// TwinCAT 3 PLC project Pushover
// Title: Pushover
// Company: Stefan Besler
// Author: Stefan Besler and contributors
// ProjectVersion: 1.1.0
// ProgramVersion: 3.1.4023.0
// libraries:
//   Tc2_Standard, * (Beckhoff Automation GmbH)
//   Tc2_System, * (Beckhoff Automation GmbH)
//   Testbench, * (Zeugwerk GmbH)
// project tree:
//   / IPushoverClient.TcIO, PushoverClient.TcPOU
//   _DataTypes/ PushoverMessageType.TcDUT, PushoverPriority.TcDUT, PushoverRequest.TcDUT, PushoverSound.TcDUT
//   _Tests/ PushoverClientTest.TcPOU

// ---- _DataTypes/PushoverMessageType.TcDUT
{attribute 'qualified_only'}
{attribute 'strict'}
TYPE PushoverMessageType :
(
	Monospace := 0,
  Html
) INT;
END_TYPE

// ---- _DataTypes/PushoverPriority.TcDUT
{attribute 'qualified_only'}
{attribute 'strict'}
TYPE PushoverPriority :
(
  /// When the priority parameter is specified with a value of -2, messages will be considered lowest priority 
  /// and will not generate any notification. On iOS, the application badge number will be increased.
	Lowest := -2,
  
  /// Messages with a priority parameter of -1 will be considered low priority and will not generate any sound 
  /// or vibration, but will still generate a popup/scrolling notification depending on the client operating system. 
  /// Messages delivered during a user's quiet hours are sent as though they had a priority of (-1).
  Low := -1,
  
  /// Messages sent without a priority parameter, or sent with the parameter set to 0, will have the default priority. 
  /// These messages trigger sound, vibration, and display an alert according to the user's device settings. 
  /// On iOS, the message will display at the top of the screen or as a modal dialog, as well as in the notification center.
  /// On Android, the message will scroll at the top of the screen and appear in the notification center.
  ///
  /// If a user has quiet hours set and your message is received during those times, your message will be delivered as though it had a priority of -1.
  Normal := 0,
  
  /// Messages sent with a priority of 1 are high priority messages that bypass a user's quiet hours.
  /// These messages will always play a sound and vibrate (if the user's device is configured to) 
  /// regardless of the delivery time. High-priority should only be used when necessary and appropriate.
  /// 
  /// High-priority messages are highlighted in red in the device clients.
  High := 1,
  
  /// Emergency-priority notifications are similar to high-priority notifications, but they are repeated until the notification 
  /// is acknowledged by the user. These are designed for dispatching and on-call situations where it is critical that a 
  /// notification be repeatedly shown to the user (or all users of the group that the message was sent to) until it is acknowledged.
  /// The first user in a group to acknowledge a message will cancel retries for all other users in the group.
  ///
  /// Applications sending emergency notifications are issued a receipt that can be used to get the status of a notification and 
  /// find out whether it was acknowledged, or automatically receive a callback when the user has acknowledged the notification. 
  ///
  /// To send an emergency-priority notification, the priority parameter must be set to 2 and the retry and expire parameters must be supplied.
  ///
  /// The retry parameter specifies how often (in seconds) the Pushover servers will send the same notification to the user. 
  /// In a situation where your user might be in a noisy environment or sleeping, retrying the notification (with sound and vibration) 
  /// will help get his or her attention. This parameter must have a value of at least 30 seconds between retries.
  ///
  /// The expire parameter specifies how many seconds your notification will continue to be retried for (every retry seconds). 
  /// If the notification has not been acknowledged in expire seconds, it will be marked as expired and will stop being sent to the user. 
  /// Note that the notification is still shown to the user after it is expired, but it will not prompt the user for acknowledgement.
  /// This parameter must have a maximum value of at most 10800 seconds (3 hours), though the total number of retries will be capped at 50 regardless of the expire parameter.
  ///
  /// For example, sending a retry parameter of 60 and an expire parameter of 1800 will cause your notification to be retried
  /// every 60 seconds for 30 minutes. A retry parameter of 30 and an expire parameter of 10800 will retry every 30 seconds up to 25 minutes due to the cap of 50 retries.
  ///
  /// The optional callback parameter may be supplied with a publicly-accessible URL that pushover servers will 
  /// send a request to when the user has acknowledged your notification.
  /// When your application sends an emergency-priority notification, pushover API will respond with a receipt value that can be used to get information about
  /// whether the notification has been acknowledged. See pushover receipts and callbacks section for more information.
  /// If your application is not capable of storing receipt identifiers, you can send a tags parameter of comma-separated, arbitrary tags 
  /// which will be stored with the receipt on pushover servers. You can then use the cancel_by_tag API call to cancel all receipts with a specific tag.
  Emergency := 2
) INT;
END_TYPE

// ---- _DataTypes/PushoverRequest.TcDUT
TYPE INTERNAL PushoverRequest :
STRUCT
  TokenLength : INT;
  UserLength : INT;
  TitleLength : INT;  
  MessageLength : INT;
  DeviceLength : INT;
  UrlLength : INT;
  UrlTitleLength : INT;
  CallbackLength : INT;  
  ProxyHostLength : INT;  
  
  Retry : INT;
  Expire : INT;  
  MessageType : PushoverMessageType;  
  Priority : PushoverPriority;
  Sound : PushoverSound;
  Timestamp : INT; //< UNIX Timestamp in seconds 
  TimeToLive : INT; //< in seconds
  ProxyPort : INT;

  Token : STRING(80);
  User : STRING(80);  
  Device : STRING(80);
  Url : STRING(511);  
  UrlTitle : STRING(99);
  Callback : STRING(255);
  ProxyHost : STRING(80);
  Title : STRING(249);  
  Message : STRING(1023);  
END_STRUCT
END_TYPE

// ---- _DataTypes/PushoverSound.TcDUT
{attribute 'qualified_only'}
{attribute 'strict'}
TYPE PushoverSound :
(
  Pushover,
  Bike,
  Bugle,
  Cashregister,
  Classical,
  Cosmic,
  Falling,
  Gamelan,
  Incoming,
  Intermission,
  Magic,
  Mechanical,
  Pianobar,
  Siren,
  Spacealarm,
  Tugboat,
  Alien,
  Climb,
  Persistent_,
  Echo,
  Updown,
  Vibrate,
  None
) INT;
END_TYPE

// ---- IPushoverClient.TcIO
INTERFACE IPushoverClient

/// \copydoc Pushover.PushoverClient#Clear
METHOD Clear : IPushoverClient
END_METHOD

/// \copydoc Pushover.PushoverClient#EnableHtml
METHOD EnableHtml : IPushoverClient
END_METHOD

/// \copydoc Pushover.PushoverClient#EnableMonospace
METHOD EnableMonospace : IPushoverClient
END_METHOD

/// \copydoc Pushover.PushoverClient#SendMessageAsync
METHOD SendMessageAsync
VAR_IN_OUT CONSTANT
  title : STRING(255);
  message : STRING(255);
END_VAR
END_METHOD

/// \copydoc Pushover.PushoverClient#WithCallback
METHOD WithCallback : IPushoverClient
VAR_IN_OUT CONSTANT
  callback : STRING(255);
END_VAR
END_METHOD

/// \copydoc Pushover.PushoverClient#WithDevice
METHOD WithDevice : IPushoverClient
VAR_IN_OUT CONSTANT
  device : STRING(80);
END_VAR
END_METHOD

/// \copydoc Pushover.PushoverClient#WithExpire
METHOD WithExpire : IPushoverClient
VAR_INPUT
  expire : INT;
END_VAR
END_METHOD

/// \copydoc Pushover.PushoverClient#WithPriority
METHOD WithPriority : IPushoverClient
VAR_INPUT
  priority : PushoverPriority;
END_VAR
END_METHOD

/// \copydoc Pushover.PushoverClient#WithProxy
METHOD WithProxy : IPushoverClient
VAR_IN_OUT CONSTANT
  host : STRING(80);
END_VAR
VAR_INPUT
  port : INT;
END_VAR
END_METHOD

/// \copydoc Pushover.PushoverClient#WithRetry
METHOD WithRetry : IPushoverClient
VAR_INPUT
  retry : INT;
END_VAR
END_METHOD

/// \copydoc Pushover.PushoverClient#WithSound
METHOD WithSound : IPushoverClient
VAR_INPUT
  sound : PushoverSound;
END_VAR
END_METHOD

/// \copydoc Pushover.PushoverClient#WithTimestamp
METHOD WithTimestamp : IPushoverClient
VAR_INPUT
  timestamp : INT; //< UNIX Timestamp in seconds
END_VAR
END_METHOD

/// \copydoc Pushover.PushoverClient#WithTimeToLive
METHOD WithTimeToLive : IPushoverClient
VAR_INPUT
  ttl : INT; //< Seconds until this message should be automatically removed from the device. Needs to be positive
END_VAR
END_METHOD

/// \copydoc Pushover.PushoverClient#WithUrl
METHOD WithUrl : IPushoverClient
VAR_IN_OUT CONSTANT
  url : STRING(255);
END_VAR
END_METHOD

/// \copydoc Pushover.PushoverClient#WithUrlTitle
METHOD WithUrlTitle : IPushoverClient
VAR_IN_OUT CONSTANT
  urlTitle : STRING(255);
END_VAR
END_METHOD

END_INTERFACE

// ---- PushoverClient.TcPOU
/// This the main class of the library. It represents a Pushover app and
/// is tied to a unique API token. When constructing the object it is mandatory to pass
/// an `app-token` as well as a `user-token`.
///
/// Here's a simple example, which sends a pushover notification to a specific device of the user.
/// Note that this class uses a fluent API to configure the properties of a notification.
/// The actual action of sending the notification is triggered by [SendMessageAsync](xref:Pushover.PushoverClient#SendMessageAsync).
/// The ´Async´ Suffix in this method indicates that this action has to be waited for by checking for ´NOT _pushoverClient.Busy´ before
/// sending another notification.
///
/// ```sti
/// PROGRAM MAIN
/// VAR
///   _send : BOOL; // boolean, which can be triggered to send a message
///   _pushoverClient : Pushover.PushoverClient('<your_pushover_apptoken>', '<your_pushover_user>'); 
/// END_VAR
/// ```
/// ```std
/// IF _send
/// THEN
///   _send := FALSE;
///   _pushoverClient
///     .SendMessageAsync('Hello World!');
/// END_IF
///
/// _pushoverClient.Cyclic();
/// ```
{attribute 'conditionalshow_all_locals'}
{attribute 'no_explicit_call' := 'This FB is a CLASS and must be accessed using methods and/or properties'}
{attribute 'hide_all_locals'}
FUNCTION_BLOCK PushoverClient IMPLEMENTS IPushoverClient
VAR
  _busy : BOOL;
  _error : BOOL;
  _errorMessage : STRING(255);
  
  _request : PushoverRequest;
  _server : Tc2_System.ADSRDWRTEX;
END_VAR
VAR CONSTANT
  _defaultHost : STRING := '127.0.0.1.1.1';
  _defaultPort : UINT := 25733;
END_VAR

/// This property can be used to check if the client is ready for sending a notification. If the client is not 
/// ready or an error occurs during sending (e.g. not internet connection, Pushover Twincat Service is not running, ...)
/// the property [Error](xref:Pushover.PushoverClient#Error) returns `true`.
{attribute 'monitoring' := 'call'}
PROPERTY Busy : BOOL
GET
Busy := _busy;
END_GET
SET // PROTECTED
_busy := Busy;

IF _busy
THEN
  _error := FALSE;
END_IF
END_SET
END_PROPERTY

/// Resets all `WithXXX` statements to their default values.
METHOD Clear : IPushoverClient
VAR
  token : STRING;
  user : STRING;
  host : STRING := '127.0.0.1.1.1';
  port : UINT := 25733;  
END_VAR
token := THIS^.Token;
user := THIS^.User;
host := THIS^.Host;
port := THIS^.Port;

Tc2_System.MEMSET(ADR(_request), 0, SIZEOF(_request));
_request.Priority := PushoverPriority.Normal;
_request.Sound := PushoverSound.Pushover;

THIS^.Token := token;
THIS^.User := user;
THIS^.Host := _defaultHost;
THIS^.Port := _defaultPort;

Clear := THIS^;
END_METHOD

/// This method has to be called cyclically and takes care of the communication with the `Pushover Twincat Service`, which is reached 
/// via [Host](xref:Pushover.PushoverClient#Host) and [Port](xref:Pushover.PushoverClient#Port).
/// You can use the properties [Busy](xref:Pushover.PushoverClient#Busy) and [Error](xref:Pushover.PushoverClient#Error) to check weather an
/// operation was successful (`NOT Busy AND NOT Error`) or failed (`Error`), respectively.
METHOD Cyclic
VAR_INST
  errorTrig : Tc2_Standard.R_TRIG;
END_VAR
IF NOT Busy
THEN
  RETURN;
END_IF

_server(IDXOFFS:=0, 
        WRITELEN:=SIZEOF(_request),
        SRCADDR:=ADR(_request),
        WRTRD:=TRUE, 
        TMOUT:=T#5S,
        ERR=>,
        BUSY=>,
        ERRID=>);
  
IF _server.ERR // fallback to proxy
THEN
  Error := TRUE;
  ErrorMessage := Tc2_Standard.CONCAT('Error Code: ', UDINT_TO_STRING(_server.ERRID));
ELSIF NOT _server.BUSY 
THEN
  Busy := FALSE;
END_IF
END_METHOD

/// Enables Monospace in the pushover message
/// Either [HTML](xref:Pushover.PushoverClient#EnableHtml) or [Monospace](xref:Pushover.PushoverClient#EnableMonspace) can be enabled
METHOD EnableHtml : IPushoverClient
_request.MessageType := PushoverMessageType.Html;

EnableHtml := THIS^;
END_METHOD

/// Enables HTML in the pushover message
/// Either [HTML](xref:Pushover.PushoverClient#EnableHtml) or [Monospace](xref:Pushover.PushoverClient#EnableMonspace) can be enabled
METHOD EnableMonospace : IPushoverClient
_request.MessageType := PushoverMessageType.Monospace;

EnableMonospace := THIS^;
END_METHOD

/// Returns `true` if any error occured when calling an `XXX_Async` method of this object. The details of the error
/// are available by checking the proeprty
{attribute 'monitoring' := 'call'}
PROPERTY Error : BOOL
GET
Error := _error;
END_GET
SET // PROTECTED
_error := Error;

IF _error
THEN
  _busy := FALSE;
END_IF
END_SET
END_PROPERTY

/// Only valid if `Error=TRUE`, returns the explanation why the call of an `XXX_Async` method failed.
{attribute 'monitoring' := 'call'}
PROPERTY ErrorMessage : STRING(255)
GET
IF _error
THEN
  ErrorMessage := _errorMessage;
END_IF
END_GET
SET // PROTECTED
_errorMessage := ErrorMessage;
END_SET
END_PROPERTY

METHOD FB_init : BOOL
VAR_INPUT
	bInitRetains : BOOL; // if TRUE, the retain variables are initialized (warm start / cold start)
	bInCopyCode : BOOL;  // if TRUE, the instance afterwards gets moved into the copy code (online change)
  
  /// The pushover API token
  token : STRING;
  
  /// The user/group key (not e-mail address) of your user (or you),
  /// viewable when logged into the [pushover dashboard](https://pushover.net/login)
  user : STRING;
END_VAR
THIS^.Token := token;
THIS^.User := user;
THIS^.Host := _defaultHost;
THIS^.Port := _defaultPort;

Clear();
END_METHOD

/// Returns the AMS Net Id of the `Pushover Twincat Service`. Defauls to localhost
PROPERTY Host : STRING
GET
Host := _server.NETID;
END_GET
SET
_server(WRTRD := FALSE,
       NETID := Host,
       BUSY=>,
       ERR=>,
       ERRID=>);
END_SET
END_PROPERTY

PROPERTY Port : UINT
GET
Port := _server.PORT;
END_GET
SET
_server(WRTRD := FALSE,
       PORT := Port,
       BUSY=>,
       ERR=>,
       ERRID=>);
END_SET
END_PROPERTY

METHOD SendMessageAsync
VAR_IN_OUT CONSTANT
  title : STRING(255);
  message : STRING(255);
END_VAR
IF NOT Busy
THEN
  _request.TitleLength := Tc2_Standard.LEN(title);
  _request.Title := title;
  _request.MessageLength := Tc2_Standard.LEN(message);
  _request.Message := message;
  
  _server(WRTRD := FALSE,
         IDXGRP:=0,
         BUSY=>,
         ERR=>,
         ERRID=>);    
  Busy := TRUE;
ELSE
  Error := TRUE;
  _errorMessage := 'Client can not executed parallel requests!';
END_IF
END_METHOD

PROPERTY Token : STRING
GET
Token := _request.Token;
END_GET
SET
_request.Token := Token;
_request.TokenLength := Tc2_Standard.LEN(_request.Token);
END_SET
END_PROPERTY

PROPERTY User : STRING
GET
User := _request.User;
END_GET
SET
_request.User := User;
_request.UserLength := Tc2_Standard.LEN(_request.User);
END_SET
END_PROPERTY

/// Callback parameter may be supplied with a publicly-accessible URL that the
/// pushover servers will send a request to when the user has acknowledged your
/// notification.
/// Only used if priority is set to emergency.
METHOD WithCallback : IPushoverClient
VAR_IN_OUT CONSTANT
  callback : STRING(255);
END_VAR
_request.CallbackLength := Tc2_Standard.LEN(callback);
_request.Callback := callback;

WithCallback := THIS^;
END_METHOD

/// Your user's device name to send the message directly to that device,
/// rather than all of the user's devices
METHOD WithDevice : IPushoverClient
VAR_IN_OUT CONSTANT
  device : STRING(80);
END_VAR
_request.DeviceLength := Tc2_Standard.LEN(device);
_request.Device := device;

WithDevice := THIS^;
END_METHOD

/// Specifies how many seconds your notification will continue to be retried for (every retry seconds).
/// Only required if priority is set to emergency.
METHOD WithExpire : IPushoverClient
VAR_INPUT
  expire : INT;
END_VAR
_request.Expire := expire;

WithExpire := THIS^;
END_METHOD

/// Priority of the message
METHOD WithPriority : IPushoverClient
VAR_INPUT
  priority : PushoverPriority;
END_VAR
_request.Priority := priority;

WithPriority := THIS^;
END_METHOD

/// Adds a ttl to the Pushover message
METHOD WithProxy : IPushoverClient
VAR_IN_OUT CONSTANT
  host : STRING(80);
END_VAR
VAR_INPUT
  port : INT;
END_VAR
_request.ProxyHostLength := Tc2_Standard.LEN(host);
_request.ProxyHost := host;
_request.ProxyPort := port;

WithProxy := THIS^;
END_METHOD

/// Specifies how often (in seconds) the Pushover servers will send the same notification to the user.
/// Only required if priority is set to emergency.
METHOD WithRetry : IPushoverClient
VAR_INPUT
  retry : INT;
END_VAR
_request.Retry := retry;

WithRetry := THIS^;
END_METHOD

/// Priority of the message
METHOD WithSound : IPushoverClient
VAR_INPUT
  sound : PushoverSound;
END_VAR
_request.Sound := sound;

WithSound := THIS^;
END_METHOD

/// A Unix timestamp of your message's date and time to display to the user,
/// rather than the time your message is received by the pushover API
METHOD WithTimestamp : IPushoverClient
VAR_INPUT
  timestamp : INT; //< UNIX Timestamp in seconds
END_VAR
_request.Timestamp := timestamp;

WithTimestamp := THIS^;
END_METHOD

/// Adds a ttl to the Pushover message
METHOD WithTimeToLive : IPushoverClient
VAR_INPUT
  ttl : INT; //< Seconds until this message should be automatically removed from the device. Needs to be positive
END_VAR
_request.TimeToLive := ttl;

WithTimeToLive := THIS^;
END_METHOD

/// A supplementary URL to show with your message
METHOD WithUrl : IPushoverClient
VAR_IN_OUT CONSTANT
  url : STRING(255);
END_VAR
_request.UrlLength := Tc2_Standard.LEN(url);
_request.Url := url;

WithUrl := THIS^;
END_METHOD

/// A title for your supplementary URL, otherwise just the URL is shown
METHOD WithUrlTitle : IPushoverClient
VAR_IN_OUT CONSTANT
  urlTitle : STRING(255);
END_VAR
_request.UrlTitleLength := Tc2_Standard.LEN(urlTitle);
_request.UrlTitle := urlTitle;

WithUrlTitle := THIS^;
END_METHOD

END_FUNCTION_BLOCK

// ---- _Tests/PushoverClientTest.TcPOU
FUNCTION_BLOCK PushoverClientTest EXTENDS PushoverClient IMPLEMENTS Testbench.IUnitTest
VAR
  _sampleRequest : PushoverRequest;
END_VAR
VAR CONSTANT
  _testAppToken : STRING := 'APP_TOKEN';
  _testUserToken : STRING := 'USER_TOKEN';
END_VAR

METHOD FB_init : BOOL
VAR_INPUT
	bInitRetains : BOOL; // if TRUE, the retain variables are initialized (warm start / cold start)
	bInCopyCode : BOOL;  // if TRUE, the instance afterwards gets moved into the copy code (online change)
  
  /// The pushover API token
  token : STRING;
  
  /// The user/group key (not e-mail address) of your user (or you),
  /// viewable when logged into the [pushover dashboard](https://pushover.net/login)
  user : STRING;
END_VAR
SUPER^.FB_init(bInitRetains, bInCopyCode, _testAppToken, _testUserToken);

_sampleRequest.TokenLength := 1;
_sampleRequest.UserLength := 2;
_sampleRequest.TitleLength := 3;
_sampleRequest.MessageLength := 4;
_sampleRequest.DeviceLength := 5;
_sampleRequest.UrlLength := 6;
_sampleRequest.UrlTitleLength := 7;
_sampleRequest.CallbackLength := 8;
_sampleRequest.ProxyHostLength := 9;
  
_sampleRequest.Token := 'token';
_sampleRequest.User := 'user';
_sampleRequest.Retry := 3;
_sampleRequest.Expire := 5;
_sampleRequest.MessageType := PushoverMessageType.Html;  
_sampleRequest.Priority := PushoverPriority.High;
_sampleRequest.Sound := PushoverSound.Cashregister;
_sampleRequest.Timestamp := 5;
_sampleRequest.TimeToLive := 50;
_sampleRequest.ProxyPort := 8080;

_sampleRequest.Title := 'Title';
_sampleRequest.Message := 'Message';
_sampleRequest.Device := 'Device';
_sampleRequest.Url := 'Url';
_sampleRequest.UrlTitle := 'UrlTitle';
_sampleRequest.Callback := 'Callback';
_sampleRequest.ProxyHost := 'ProxyHost';
END_METHOD

METHOD SendMessageAsync
VAR_IN_OUT CONSTANT
  title : STRING(255);
  message : STRING(255);
END_VAR
IF NOT Busy
THEN
  _request.TitleLength := Tc2_Standard.LEN(title);
  _request.Title := title;
  _request.MessageLength := Tc2_Standard.LEN(message);
  _request.Message := message;
  
  _server(WRTRD := FALSE,
         IDXGRP:=0,
         BUSY=>,
         ERR=>,
         ERRID=>);    
  Busy := TRUE;
ELSE
  Error := TRUE;
  ErrorMessage := 'Client can not executed parallel requests!';
END_IF
END_METHOD

METHOD Test_Busy
VAR_INPUT
  assertions : Testbench.IAssertions;
END_VAR
Error := TRUE;

Busy := TRUE;

assertions.IsFalse(Error, '');
assertions.IsTrue(Busy, '');
END_METHOD

METHOD Test_Clear
VAR_INPUT
  assertions : Testbench.IAssertions;
END_VAR
_request := _sampleRequest;
_request.Token := _testAppToken;
_request.User := _testUserToken;

Clear();

assertions.EqualsString('', _request.Url, 'Url is reset');
assertions.EqualsString('', _request.UrlTitle, 'UrlTitle is reset');
assertions.EqualsString('', _request.Message, 'Message is reset');
assertions.EqualsString('', _request.Title, 'Title is reset');
assertions.EqualsInt(0, _request.Retry, 'Retry is reset');
assertions.EqualsString(_testAppToken, Token, 'Token is initialized with APP_TOKEN');
assertions.EqualsString(_testUserToken, User, 'User is initialized with USER_TOKEN');
assertions.EqualsString(_defaultHost, Host, 'Host is initialized with the default');
assertions.EqualsUint(_defaultPort, Port, 'Port is initialized with the default');
assertions.EqualsInt(PushoverPriority.Normal, _request.Priority, 'The default value of priority is normal');
assertions.EqualsInt(PushoverSound.Pushover, _request.Sound, 'The default sund is pushover');
END_METHOD

METHOD Test_Defaults
VAR_INPUT
  assertions : Testbench.IAssertions;
END_VAR
assertions.EqualsString(_testAppToken, Token, 'Token is initialized with APP_TOKEN');
assertions.EqualsString(_testUserToken, User, 'User is initialized with USER_TOKEN');
assertions.EqualsString(_defaultHost, Host, 'Host is initialized with the default');
assertions.EqualsUint(_defaultPort, Port, 'Port is initialized with the default');
assertions.IsFalse(Busy, 'Object is not busy');
assertions.IsFalse(Error, 'Object has not error');
assertions.EqualsInt(PushoverPriority.Normal, _request.Priority, 'The default value of priority is normal');
assertions.EqualsInt(PushoverSound.Pushover, _request.Sound, 'The default sund is pushover');
END_METHOD

METHOD Test_EnableHtml
VAR_INPUT
  assertions : Testbench.IAssertions;
END_VAR
VAR_INST
  self : IPushoverClient := THIS^;
  intrf : IPushoverClient;
END_VAR
_request := _sampleRequest;

intrf := EnableHtml();

assertions.EqualsInt(PushoverMessageType.Html, _request.MessageType, '');
assertions.IsTrue(self = intrf, '');
END_METHOD

METHOD Test_EnableMonospace
VAR_INPUT
  assertions : Testbench.IAssertions;
END_VAR
VAR_INST
  self : IPushoverClient := THIS^;
  intrf : IPushoverClient;
END_VAR
_request := _sampleRequest;

intrf := EnableMonospace();

assertions.EqualsInt(PushoverMessageType.Monospace, _request.MessageType, '');
assertions.IsTrue(self = intrf, '');
END_METHOD

METHOD Test_Error
VAR_INPUT
  assertions : Testbench.IAssertions;
END_VAR
Busy := TRUE;

Error := TRUE;

assertions.IsFalse(Busy, '');
assertions.IsTrue(Error, '');
END_METHOD

METHOD Test_WithCallback
VAR_INPUT
  assertions : Testbench.IAssertions;
END_VAR
VAR_INST
  self : IPushoverClient := THIS^;
  intrf : IPushoverClient;
END_VAR
_request := _sampleRequest;

intrf := WithCallback('xyz');

assertions.EqualsInt(3, _request.CallbackLength, '');
assertions.EqualsString('xyz', _request.Callback, '');
assertions.IsTrue(self = intrf, '');
END_METHOD

METHOD Test_WithDevice
VAR_INPUT
  assertions : Testbench.IAssertions;
END_VAR
VAR_INST
  self : IPushoverClient := THIS^;
  intrf : IPushoverClient;
END_VAR
_request := _sampleRequest;

intrf := WithDevice('xyz');

assertions.EqualsInt(3, _request.DeviceLength, '');
assertions.EqualsString('xyz', _request.Device, '');
assertions.IsTrue(self = intrf, '');
END_METHOD

METHOD Test_WithExpire
VAR_INPUT
  assertions : Testbench.IAssertions;
END_VAR
VAR_INST
  self : IPushoverClient := THIS^;
  intrf : IPushoverClient;
END_VAR
_request := _sampleRequest;

intrf := WithExpire(115);

assertions.EqualsInt(115, _request.Expire, '');
assertions.IsTrue(self = intrf, '');
END_METHOD

METHOD Test_WithPriority
VAR_INPUT
  assertions : Testbench.IAssertions;
END_VAR
VAR_INST
  self : IPushoverClient := THIS^;
  intrf : IPushoverClient;
END_VAR
_request := _sampleRequest;

intrf := WithPriority(PushoverPriority.Lowest);

assertions.EqualsInt(PushoverPriority.Lowest, _request.Priority, '');
assertions.IsTrue(self = intrf, '');
END_METHOD

METHOD Test_WithProxy
VAR_INPUT
  assertions : Testbench.IAssertions;
END_VAR
VAR_INST
  self : IPushoverClient := THIS^;
  intrf : IPushoverClient;
END_VAR
_request := _sampleRequest;

intrf := WithProxy('xyz', 8989);

assertions.EqualsInt(8989, _request.ProxyPort, '');
assertions.EqualsInt(3, _request.ProxyHostLength, '');
assertions.EqualsString('xyz', _request.ProxyHost, '');
assertions.IsTrue(self = intrf, '');
END_METHOD

METHOD Test_WithRetry
VAR_INPUT
  assertions : Testbench.IAssertions;
END_VAR
VAR_INST
  self : IPushoverClient := THIS^;
  intrf : IPushoverClient;
END_VAR
_request := _sampleRequest;

intrf := WithRetry(115);

assertions.EqualsInt(115, _request.Retry, '');
assertions.IsTrue(self = intrf, '');
END_METHOD

METHOD Test_WithSound
VAR_INPUT
  assertions : Testbench.IAssertions;
END_VAR
VAR_INST
  self : IPushoverClient := THIS^;
  intrf : IPushoverClient;
END_VAR
_request := _sampleRequest;

intrf := WithSound(PushoverSound.Cosmic);

assertions.EqualsInt(PushoverSound.Cosmic, _request.Sound, '');
assertions.IsTrue(self = intrf, '');
END_METHOD

METHOD Test_WithTimestamp
VAR_INPUT
  assertions : Testbench.IAssertions;
END_VAR
VAR_INST
  self : IPushoverClient := THIS^;
  intrf : IPushoverClient;
END_VAR
_request := _sampleRequest;

intrf := WithTimestamp(115);

assertions.EqualsInt(115, _request.Timestamp, '');
assertions.IsTrue(self = intrf, '');
END_METHOD

METHOD Test_WithTimeToLive
VAR_INPUT
  assertions : Testbench.IAssertions;
END_VAR
VAR_INST
  self : IPushoverClient := THIS^;
  intrf : IPushoverClient;
END_VAR
_request := _sampleRequest;

intrf := WithTimeToLive(115);

assertions.EqualsInt(115, _request.TimeToLive, '');
assertions.IsTrue(self = intrf, '');
END_METHOD

METHOD Test_WithUrl
VAR_INPUT
  assertions : Testbench.IAssertions;
END_VAR
VAR_INST
  self : IPushoverClient := THIS^;
  intrf : IPushoverClient;
END_VAR
_request := _sampleRequest;

intrf := WithUrl('xyz');

assertions.EqualsInt(3, _request.UrlLength, '');
assertions.EqualsString('xyz', _request.Url, '');
assertions.IsTrue(self = intrf, '');
END_METHOD

METHOD Test_WithUrlTitle
VAR_INPUT
  assertions : Testbench.IAssertions;
END_VAR
VAR_INST
  self : IPushoverClient := THIS^;
  intrf : IPushoverClient;
END_VAR
_request := _sampleRequest;

intrf := WithUrlTitle('xyz');

assertions.EqualsInt(3, _request.UrlTitleLength, '');
assertions.EqualsString('xyz', _request.UrlTitle, '');
assertions.IsTrue(self = intrf, '');
END_METHOD

END_FUNCTION_BLOCK
